//-----------------------------------------------------------------------------------------------------------------
// ExternControl: EXT_MOTION_CONTROL
//
// BASIC EXAMPLE for controlling PLC_MOTION_LAYER
//-----------------------------------------------------------------------------------------------------------------
PROGRAM MAIN
VAR
  //---------------------------------------------------------------------------------------------------------------
  eInitPlcMotion  AT %I*  : E_PROGRESS;   // startup indicator from PLC_MOTION plc
  //---------------------------------------------------------------------------------------------------------------

  nAxis           : UINT := 1;  // you choose

  bStartAxis,
  bStartCam       : BOOL;

  eStateAxis,
  eStateCam       : E_PROGRESS;

  eCtrlFunction   : E_AXIS_CTRL   := E_AXIS_CTRL.AXIS_ENABLE;   // for you to set
  eStateFunction  : E_AXIS_STATE  := E_AXIS_STATE.AXIS_ENABLE;  // for you to set so the result can be checked correctly

  stMsg           : ST_Message;
  eMsgState       : e_message_state;
  eMsgProgress    : E_PROGRESS;
END_VAR

//-----------------------------------------------------------------------------------------------------------------
// Local time; used for timestamps
//-----------------------------------------------------------------------------------------------------------------
GVL_MSG.fbLocalTime(
                    sLocalTime                => GVL_MSG.sLocalTime, 
                    dtLocalTime               => GVL_MSG.dtLocalTime);
//-----------------------------------------------------------------------------------------------------------------
//-----------------------------------------------------------------------------------------------------------------
// PLC_MOTION_LAYER startup check: 
//  - you may evaluate this on your own terms
//  - putting it here was convenient for me in the context of this simple example
//-----------------------------------------------------------------------------------------------------------------
//-----------------------------------------------------------------------------------------------------------------
IF NOT (eInitPlcMotion = E_PROGRESS.PROGRESS_DONE)
THEN
  RETURN;
END_IF
//-----------------------------------------------------------------------------------------------------------------
//-----------------------------------------------------------------------------------------------------------------
// BASIC SEQUENCE for controlling PLC_MOTION_LAYER
//-----------------------------------------------------------------------------------------------------------------
//-----------------------------------------------------------------------------------------------------------------
TEST();
//-----------------------------------------------------------------------------------------------------------------
//-----------------------------------------------------------------------------------------------------------------
// BASIC EXAMPLE for controlling PLC_MOTION_LAYER
//-----------------------------------------------------------------------------------------------------------------
//-----------------------------------------------------------------------------------------------------------------
//-----------------------------------------------------------------------------------------------------------------
// HOW to... PtP axis
//  - you have to use the data and parameter fields in the matching GVL
//-----------------------------------------------------------------------------------------------------------------
IF NOT bStartAxis
THEN
  // this is for cleaning up your state machine
  eStateAxis                      := E_PROGRESS.PROGRESS_INIT;
END_IF
//-----------------------------------------------------------------------------------------------------------------
//-----------------------------------------------------------------------------------------------------------------
CASE eStateAxis 
OF
  E_PROGRESS.PROGRESS_INIT:
    IF bStartAxis                 // do not forget to set the motion data for the chosen axis, GVL_AXIS.Data etc. 
    THEN
      GVL_AXIS.Ctrl[nAxis].eCmd   := eCtrlFunction;

      eStateAxis                  := E_PROGRESS.PROGRESS_BUSY;
    END_IF


  E_PROGRESS.PROGRESS_BUSY:
    IF (GVL_AXIS.State[nAxis].eState = eStateFunction + E_PROGRESS.PROGRESS_DONE)
    THEN
      eStateAxis                  := E_PROGRESS.PROGRESS_DONE;

    ELSIF (GVL_AXIS.State[nAxis].eState = eStateFunction + E_PROGRESS.PROGRESS_ERROR)
    THEN
      eStateAxis                  := E_PROGRESS.PROGRESS_ERROR;
    END_IF
END_CASE
//-----------------------------------------------------------------------------------------------------------------
//-----------------------------------------------------------------------------------------------------------------
// HOW to... CAM axis
//  - you have to use the data and parameter fields in the matching GVL
//-----------------------------------------------------------------------------------------------------------------
IF NOT bStartCam
THEN
  // this is for cleaning up your state machine
  eStateCam                       := E_PROGRESS.PROGRESS_INIT;
END_IF
//-----------------------------------------------------------------------------------------------------------------
//-----------------------------------------------------------------------------------------------------------------
CASE eStateCam
OF
  E_PROGRESS.PROGRESS_INIT:
    IF bStartCam                 // do not forget to set the motion data for the chosen axis, GVL_AXIS.Data etc. 
    THEN
      GVL_CAM.Ctrl[nAxis].eCmd    := eCtrlFunction;

      eStateCam                   := E_PROGRESS.PROGRESS_BUSY;
    END_IF


  E_PROGRESS.PROGRESS_BUSY:
    IF (GVL_AXIS.State[nAxis].eState = eStateFunction + E_PROGRESS.PROGRESS_DONE)
    THEN
      eStateCam                   := E_PROGRESS.PROGRESS_DONE;

    ELSIF (GVL_AXIS.State[nAxis].eState = eStateFunction + E_PROGRESS.PROGRESS_ERROR)
    THEN
      eStateCam                   := E_PROGRESS.PROGRESS_ERROR;
    END_IF
END_CASE
//-----------------------------------------------------------------------------------------------------------------
//-----------------------------------------------------------------------------------------------------------------
//-----------------------------------------------------------------------------------------------------------------
//  /logging
//    - all life is problem solving
//-----------------------------------------------------------------------------------------------------------------
GVL_MSG.MotionMessageData.Ctrl                REF= GVL_MSG.MotionMessageCtrl;
GVL_MSG.MotionMessageData.State               REF= GVL_MSG.MotionMessageState;

GVL_MSG.MotionMessageData.MessageIndex        REF= GVL_MSG.MessageMotionIndex;
GVL_MSG.MotionMessageData.ErrorIndex          REF= GVL_MSG.MessageMotionError;

GVL_MSG.MotionMessageData.DirRoot             :=   ADR(GVL_MSG.LOG_DIR);
GVL_MSG.MotionMessageData.FileRoot            :=   ADR(GVL_MSG.LOG_FILE);

GVL_MSG.MotionMessageData.MsgList             :=   ADR(GVL_MSG.MotionMessages);
GVL_MSG.MotionMessageData.LocalTime           :=   ADR(GVL_MSG.dtLocalTime);

GVL_MSG.MotionMessageData();               

eMsgState                                     :=   f_GetState   (GVL_MSG.MotionMessageState.State);
eMsgProgress                                  :=   f_GetProgress(GVL_MSG.MotionMessageState.State);

CASE eMsgState
OF
  E_MESSAGE_STATE.MSG_STATE_NULL:
    CASE eMsgProgress
    OF
      E_PROGRESS.PROGRESS_INVALID,
      E_PROGRESS.PROGRESS_DONE:
        IF (GVL_MSG.MessageMotionIndex > GVL_MSG.MAX_MESSAGE/100) OR
           (GVL_MSG.MessageMotionError > 0)
        THEN
          GVL_MSG.MotionMessageCtrl.Cmd       := E_MESSAGE_CTRL.MSG_CTRL_WRITE;
        END_IF
    END_CASE

  E_MESSAGE_STATE.MSG_STATE_WRITE:
    CASE eMsgProgress
    OF
      E_PROGRESS.PROGRESS_ERROR,
      E_PROGRESS.PROGRESS_DONE:
        GVL_MSG.MotionMessageCtrl.Cmd         := E_MESSAGE_CTRL.MSG_CTRL_NULL;
    END_CASE

ELSE
    CASE eMsgProgress
    OF
      E_PROGRESS.PROGRESS_DONE:
        GVL_MSG.MotionMessageCtrl.Cmd         := E_MESSAGE_CTRL.MSG_CTRL_NULL;
    END_CASE
END_CASE
//-----------------------------------------------------------------------------------------------------------------
//  logging/
//-----------------------------------------------------------------------------------------------------------------
//-----------------------------------------------------------------------------------------------------------------

END_PROGRAM

(* stored: Version 1.1.0.1
   POU MAIN: Id {9bc05cf8-27df-4baf-8c2e-8597e29fd5e7}, SpecialFunc None *)
